Omron Sysmac Studio project Colorificio_End_Release (Sysmac Studio 1.30.0.17, StandardProject)
(* Comment update *)

# Controller PLC: NX1P2-9024DT1 version 1.40
Task PrimaryTask (priority 4, period or condition 2000): Program0
Library OmronLib_WC_Toolbox_V1_0 1.0.0 (contents left out)

TYPE S_Colori : STRUCT
    ALPHA : INT;
    RED : INT;
    GREEN : INT;
    BLU : INT;
    NOME : STRING[256];
END_STRUCT END_TYPE

VAR_GLOBAL
    SB0 : BOOL := False;  (* pulsante avvio ciclo automatico (NA); at BuiltInIO://cpu/#0/Input_Bit_00 *)
    SB1 : BOOL := True;  (* pulsante arresto ciclo automatico (NC); at BuiltInIO://cpu/#0/Input_Bit_01 *)
    SBE : BOOL := True;  (* pulsante arresto di emergenza (NC); at BuiltInIO://cpu/#0/Input_Bit_02 *)
    YVA : BOOL;  (* libera caricatore seconda latta (A-); at BuiltInIO://cpu/#0/Output_Bit_00 *)
    YVB : BOOL;  (* libera caricatore prima latta (B-); at BuiltInIO://cpu/#0/Output_Bit_01 *)
    YVC : BOOL;  (* scarico bilancia (C+); at BuiltInIO://cpu/#0/Output_Bit_02 *)
    KM1 : BOOL;  (* motore primo nastro; at BuiltInIO://cpu/#0/Output_Bit_09 *)
    KM2 : BOOL;  (* motore secondo nastro; at IOBus://unit#3/Output Bit 8 bits/Output Bit 00 *)
    YVD : BOOL;  (* scarico coperchiatrice (D+); at BuiltInIO://cpu/#0/Output_Bit_03 *)
    a0 : BOOL := False;  (* caricatore seconda latta libero (NA); at BuiltInIO://cpu/#0/Input_Bit_03 *)
    a1 : BOOL := True;  (* caricatore seconda latta bloccato (NA); at BuiltInIO://cpu/#0/Input_Bit_04 *)
    b0 : BOOL := False;  (* caricatore prima latta libero (NA); at BuiltInIO://cpu/#0/Input_Bit_05 *)
    b1 : BOOL := True;  (* caricatore prima latta bloccato (NA); at BuiltInIO://cpu/#0/Input_Bit_06 *)
    c0 : BOOL := True;  (* scaricatore bilancia rientrato (NA); at BuiltInIO://cpu/#0/Input_Bit_07 *)
    c1 : BOOL := False;  (* scaricatore bilancia esteso (NA); at BuiltInIO://cpu/#0/Input_Bit_08 *)
    d0 : BOOL := True;  (* scaricatore coperchiatrice rientrato (NA); at BuiltInIO://cpu/#0/Input_Bit_09 *)
    d1 : BOOL := False;  (* scaricatore coperchiatrice esteso (NA); at BuiltInIO://cpu/#0/Input_Bit_10 *)
    BIL : REAL;  (* bilancia/cella di carico (Grammi) *)
    YVBASE : BOOL;  (* eroga colorante base; at BuiltInIO://cpu/#0/Output_Bit_04 *)
    YVRED : BOOL;  (* eroga colorante rosso; at BuiltInIO://cpu/#0/Output_Bit_05 *)
    YVGREEN : BOOL;  (* eroga colorante verde; at BuiltInIO://cpu/#0/Output_Bit_06 *)
    YVBLU : BOOL;  (* eroga colorante blu; at BuiltInIO://cpu/#0/Output_Bit_07 *)
    YVSCARICO : BOOL;  (* eroga totale colore; at BuiltInIO://cpu/#0/Output_Bit_08 *)
    Tbase : TIME;  (* tempo carico base *)
    Trosso : TIME;  (* tempo carico rosso *)
    Tgreen : TIME;  (* tempo carico verde *)
    Tblu : TIME;  (* tempo carico blu *)
    BLW : BOOL := True;  (* livello riserva Base White (NA); at BuiltInIO://cpu/#0/Input_Bit_11 *)
    BLR : BOOL := True;  (* livello riserva Red (NA); at BuiltInIO://cpu/#0/Input_Bit_12 *)
    BLG : BOOL := True;  (* livello riserva Green (NA); at BuiltInIO://cpu/#0/Input_Bit_13 *)
    BLB : BOOL := True;  (* livello riserva Blu (NA); at IOBus://unit#1/Input Bit 8 bits/Input Bit 00 *)
    BC1 : BOOL := False;  (* presenza seconda latta sul caricatore (NA); at IOBus://unit#1/Input Bit 8 bits/Input Bit 03 *)
    BBIL : BOOL := False;  (* presenza sulla bilancia (NA); at IOBus://unit#1/Input Bit 8 bits/Input Bit 01 *)
    BCOP : BOOL := False;  (* presenza sulla coperchiatrice (NA); at IOBus://unit#1/Input Bit 8 bits/Input Bit 04 *)
    RichiestaValvolaBase : BOOL;  (* Devo aprire la valvola della Base? *)
    RichiestaValvolaRosso : BOOL;  (* Devo aprire la valvola del Rosso? *)
    RichiestaValvolaVerde : BOOL;  (* Devo aprire la valvola del Verde? *)
    RichiestaValvolaBlu : BOOL;  (* Devo aprire la valvola del Blu? *)
    RichiestaValvolaTramoggia : BOOL;  (* Devo aprire la valvola della Tramoggia? *)
    LevelToEjectBase : REAL := -1;  (* Quantità di base da far uscire *)
    LevelToEjectRosso : REAL := -1;  (* Quantità di rosso da far uscire *)
    LevelToEjectVerde : REAL := -1;  (* Quantità di verde da far uscire *)
    LevelToEjectBlu : REAL := -1;  (* Quantità di blu da far uscire *)
    ColorDone : BOOL := False;  (* Processo di riempimento del barattolo completo *)
    PHL_RiservaBase : BOOL;  (* Lampada mancanza di base; at IOBus://unit#3/Output Bit 8 bits/Output Bit 01 *)
    PHL_RiservaRosso : BOOL;  (* Lampada mancanza di rosso; at IOBus://unit#3/Output Bit 8 bits/Output Bit 02 *)
    PHL_RiservaVerde : BOOL;  (* Lampada mancanza di verde; at IOBus://unit#3/Output Bit 8 bits/Output Bit 03 *)
    PHL_RiservaBlu : BOOL;  (* Lampada mancanza di blu; at IOBus://unit#3/Output Bit 8 bits/Output Bit 04 *)
    PHL_YVScarico : BOOL;  (* Lampada valvola tramoggia aperta; at IOBus://unit#3/Output Bit 8 bits/Output Bit 05 *)
    PHL_KM : BOOL;  (* Lampada nastri in movimento; at IOBus://unit#3/Output Bit 8 bits/Output Bit 06 *)
    PHL_Emergenza : BOOL;  (* Lampada pulsante emergenza attivato; at IOBus://unit#3/Output Bit 8 bits/Output Bit 07 *)
    LivelloTramoggia : REAL := 0.0;
    PesoTramoggia : REAL := 0.0;
    BC0 : BOOL := False;  (* presenza prima latta sul caricatore (NA); at IOBus://unit#1/Input Bit 8 bits/Input Bit 02 *)
END_VAR

PROGRAM Program0
VAR
    TimerBase : TP;
    TimerRosso : TP;
    TimerVerde : TP;
    TimerBlu : TP;
    estimatedBase : TIME;
    estimatedRosso : TIME;
    estimatedVerde : TIME;
    estimatedBlu : TIME;
    Rosso : BOOL;
    Base : BOOL;
    Verde : BOOL;
    Blu : BOOL;
    Scarico : BOOL;
    estimatedScarico : TIME;
    Tscarico : TIME;  (* Tempo di uscita del contenuto della tramoggia *)
    TimerScarico : TP;
    AspettaSvuotamentoBlu : TP;
    AspettaSvuotamentoBlu1 : TON;
    estimatedSvuotamentoBlu : TIME;
    estimatedSvuotamentoBlu1 : TIME;
    AspettaSvuotamentoScarico : TP;
    estimatedSvuotamentoScarico : TIME;
    AspettaSvuotamentoScarico1 : TON;
    estimatedSvuotamentoScarico1 : TIME;
    DelayBase : TON;  (* Attivazione base in ritardo *)
    estimatedActValvolaBase : TIME;  (* Tempo rimanente all'attivazione della valvola della base *)
    Basse : BOOL;
END_VAR
VAR_EXTERNAL
    SB1 : BOOL;
    KM1 : BOOL;
    YVC : BOOL;
    BBIL : BOOL;
    c0 : BOOL;
    c1 : BOOL;
    KM2 : BOOL;
    SB0 : BOOL;
    SBE : BOOL;
    BIL : REAL;
    RichiestaValvolaBase : BOOL;
    RichiestaValvolaRosso : BOOL;
    RichiestaValvolaVerde : BOOL;
    RichiestaValvolaBlu : BOOL;
    YVBASE : BOOL;
    YVRED : BOOL;
    YVGREEN : BOOL;
    YVBLU : BOOL;
    Tbase : TIME;
    Trosso : TIME;
    Tgreen : TIME;
    Tblu : TIME;
    RichiestaValvolaTramoggia : BOOL;
    YVSCARICO : BOOL;
    ColorDone : BOOL;  (* Processo di riempimento del barattolo completo *)
    PHL_KM : BOOL;
    PHL_Emergenza : BOOL;
    PHL_YVScarico : BOOL;
    LevelToEjectBlu : REAL;
    LevelToEjectVerde : REAL;
    LevelToEjectRosso : REAL;
    LevelToEjectBase : REAL;
    LivelloTramoggia : REAL;
    PesoTramoggia : REAL;
    PHL_RiservaBase : BOOL;
    PHL_RiservaBlu : BOOL;
    PHL_RiservaVerde : BOOL;
    PHL_RiservaRosso : BOOL;
    BLB : BOOL;
    BLR : BOOL;
    BLW : BOOL;
    BLG : BOOL;
    BCOP : BOOL;
END_VAR
VAR
    _p1 : BOOL;
    _p2 : BOOL;
    _p3 : BOOL;
    _p4 : BOOL;
    _p5 : BOOL;
    _p6 : BOOL;
    _p7 : BOOL;
    _p8 : BOOL;
    _e9 : F_TRIG;
END_VAR

(* Section Section0: ladder, written here as Structured Text *)

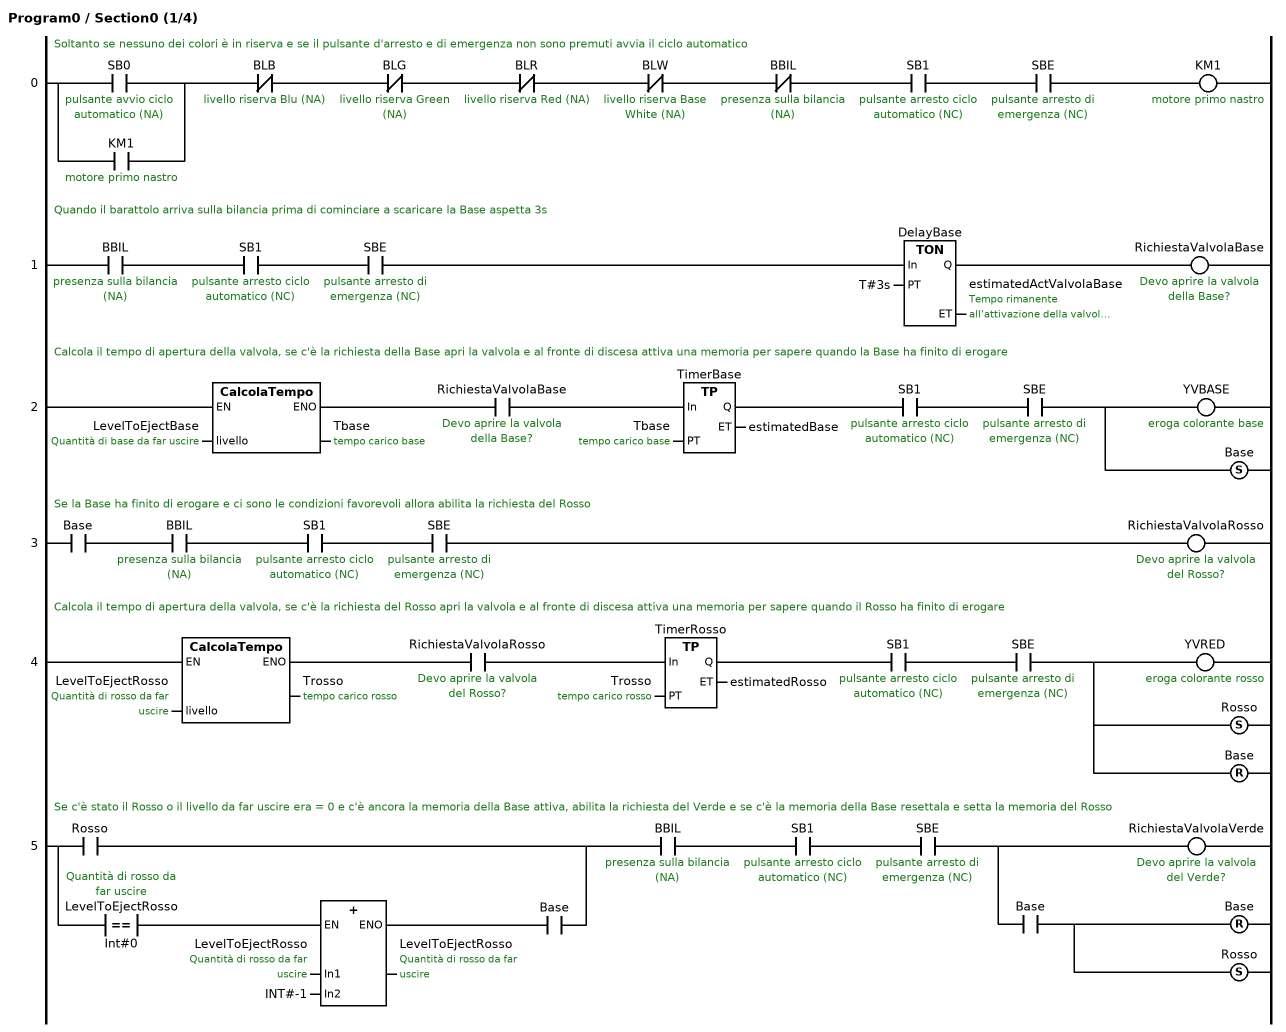
(* Rung 0: Soltanto se nessuno dei colori è in riserva e se il pulsante d'arresto e di emergenza non sono premuti avvia il ciclo automatico *)
KM1 := (SB0 OR KM1) AND NOT BLB AND NOT BLG AND NOT BLR AND NOT BLW AND NOT BBIL AND SB1 AND SBE;
(* Rung 1: Quando il barattolo arriva sulla bilancia prima di cominciare a scaricare la Base aspetta 3s *)
DelayBase(In := BBIL AND SB1 AND SBE, PT := T#3s, ET => estimatedActValvolaBase);
RichiestaValvolaBase := DelayBase.Q;
(* Rung 2: Calcola il tempo di apertura della valvola, se c'è la richiesta della Base apri la valvola e al fronte di discesa attiva una memoria per sapere quando la Base ha finito di erogare *)
Tbase := CalcolaTempo(livello := LevelToEjectBase);
TimerBase(In := RichiestaValvolaBase, PT := Tbase, ET => estimatedBase);
YVBASE := TimerBase.Q AND SB1 AND SBE;
IF TimerBase.Q AND SB1 AND SBE THEN Base := TRUE; END_IF;
(* Rung 3: Se la Base ha finito di erogare e ci sono le condizioni favorevoli allora abilita la richiesta del Rosso *)
RichiestaValvolaRosso := Base AND BBIL AND SB1 AND SBE;
(* Rung 4: Calcola il tempo di apertura della valvola, se c'è la richiesta del Rosso apri la valvola e al fronte di discesa attiva una memoria per sapere quando il Rosso ha finito di erogare *)
Trosso := CalcolaTempo(livello := LevelToEjectRosso);
TimerRosso(In := RichiestaValvolaRosso, PT := Trosso, ET => estimatedRosso);
YVRED := TimerRosso.Q AND SB1 AND SBE;
IF TimerRosso.Q AND SB1 AND SBE THEN
    Rosso := TRUE;
    Base := FALSE;
END_IF;
(* Rung 5: Se c'è stato il Rosso o il livello da far uscire era = 0 e c'è ancora la memoria della Base attiva, abilita la richiesta del Verde e se c'è la memoria della Base resettala e setta la memoria del Rosso *)
_p1 := LevelToEjectRosso = Int#0;
IF _p1 THEN LevelToEjectRosso := LevelToEjectRosso + (INT#-1); END_IF;
_p2 := (Rosso OR (_p1 AND Base)) AND BBIL AND SB1 AND SBE;
RichiestaValvolaVerde := _p2;
_p3 := _p2 AND Base;
IF _p3 THEN
    Base := FALSE;
    Rosso := TRUE;
END_IF;

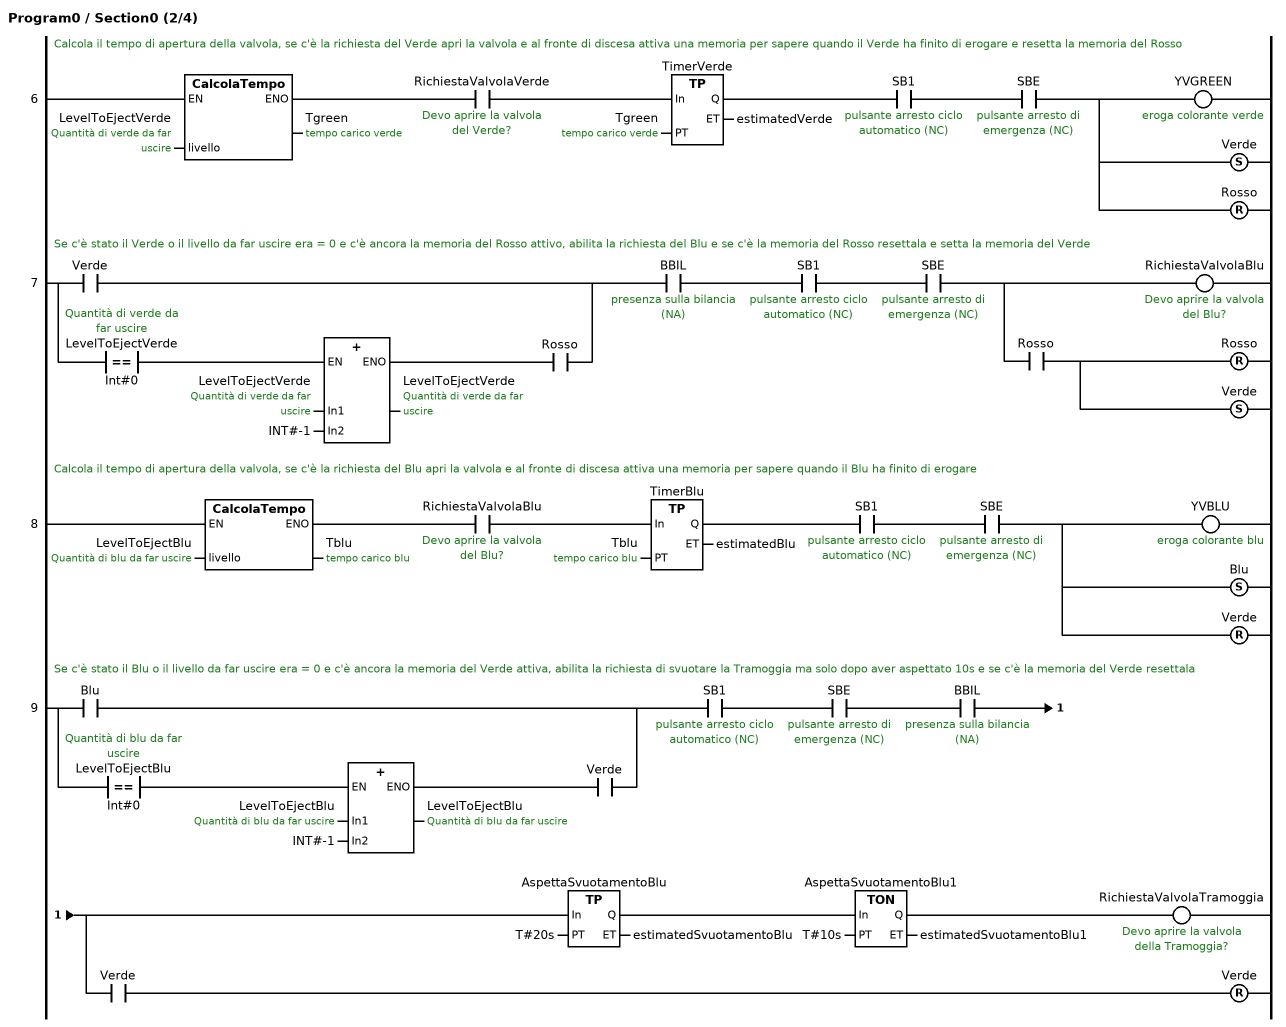
(* Rung 6: Calcola il tempo di apertura della valvola, se c'è la richiesta del Verde apri la valvola e al fronte di discesa attiva una memoria per sapere quando il Verde ha finito di erogare e resetta la memoria del Rosso *)
Tgreen := CalcolaTempo(livello := LevelToEjectVerde);
TimerVerde(In := RichiestaValvolaVerde, PT := Tgreen, ET => estimatedVerde);
YVGREEN := TimerVerde.Q AND SB1 AND SBE;
IF TimerVerde.Q AND SB1 AND SBE THEN
    Verde := TRUE;
    Rosso := FALSE;
END_IF;
(* Rung 7: Se c'è stato il Verde o il livello da far uscire era = 0 e c'è ancora la memoria del Rosso attivo, abilita la richiesta del Blu e se c'è la memoria del Rosso resettala e setta la memoria del Verde *)
_p4 := LevelToEjectVerde = Int#0;
IF _p4 THEN LevelToEjectVerde := LevelToEjectVerde + (INT#-1); END_IF;
_p5 := (Verde OR (_p4 AND Rosso)) AND BBIL AND SB1 AND SBE;
RichiestaValvolaBlu := _p5;
_p6 := _p5 AND Rosso;
IF _p6 THEN
    Rosso := FALSE;
    Verde := TRUE;
END_IF;
(* Rung 8: Calcola il tempo di apertura della valvola, se c'è la richiesta del Blu apri la valvola e al fronte di discesa attiva una memoria per sapere quando il Blu ha finito di erogare *)
Tblu := CalcolaTempo(livello := LevelToEjectBlu);
TimerBlu(In := RichiestaValvolaBlu, PT := Tblu, ET => estimatedBlu);
YVBLU := TimerBlu.Q AND SB1 AND SBE;
IF TimerBlu.Q AND SB1 AND SBE THEN
    Blu := TRUE;
    Verde := FALSE;
END_IF;
(* Rung 9: Se c'è stato il Blu o il livello da far uscire era = 0 e c'è ancora la memoria del Verde attiva, abilita la richiesta di svuotare la Tramoggia ma solo dopo aver aspettato 10s e se c'è la memoria del Verde resettala *)
_p7 := LevelToEjectBlu = Int#0;
IF _p7 THEN LevelToEjectBlu := LevelToEjectBlu + (INT#-1); END_IF;
_p8 := (Blu OR (_p7 AND Verde)) AND SB1 AND SBE AND BBIL;
AspettaSvuotamentoBlu(In := _p8, PT := T#20s, ET => estimatedSvuotamentoBlu);
AspettaSvuotamentoBlu1(In := AspettaSvuotamentoBlu.Q, PT := T#10s, ET => estimatedSvuotamentoBlu1);
RichiestaValvolaTramoggia := AspettaSvuotamentoBlu1.Q;
IF _p8 AND Verde THEN Verde := FALSE; END_IF;

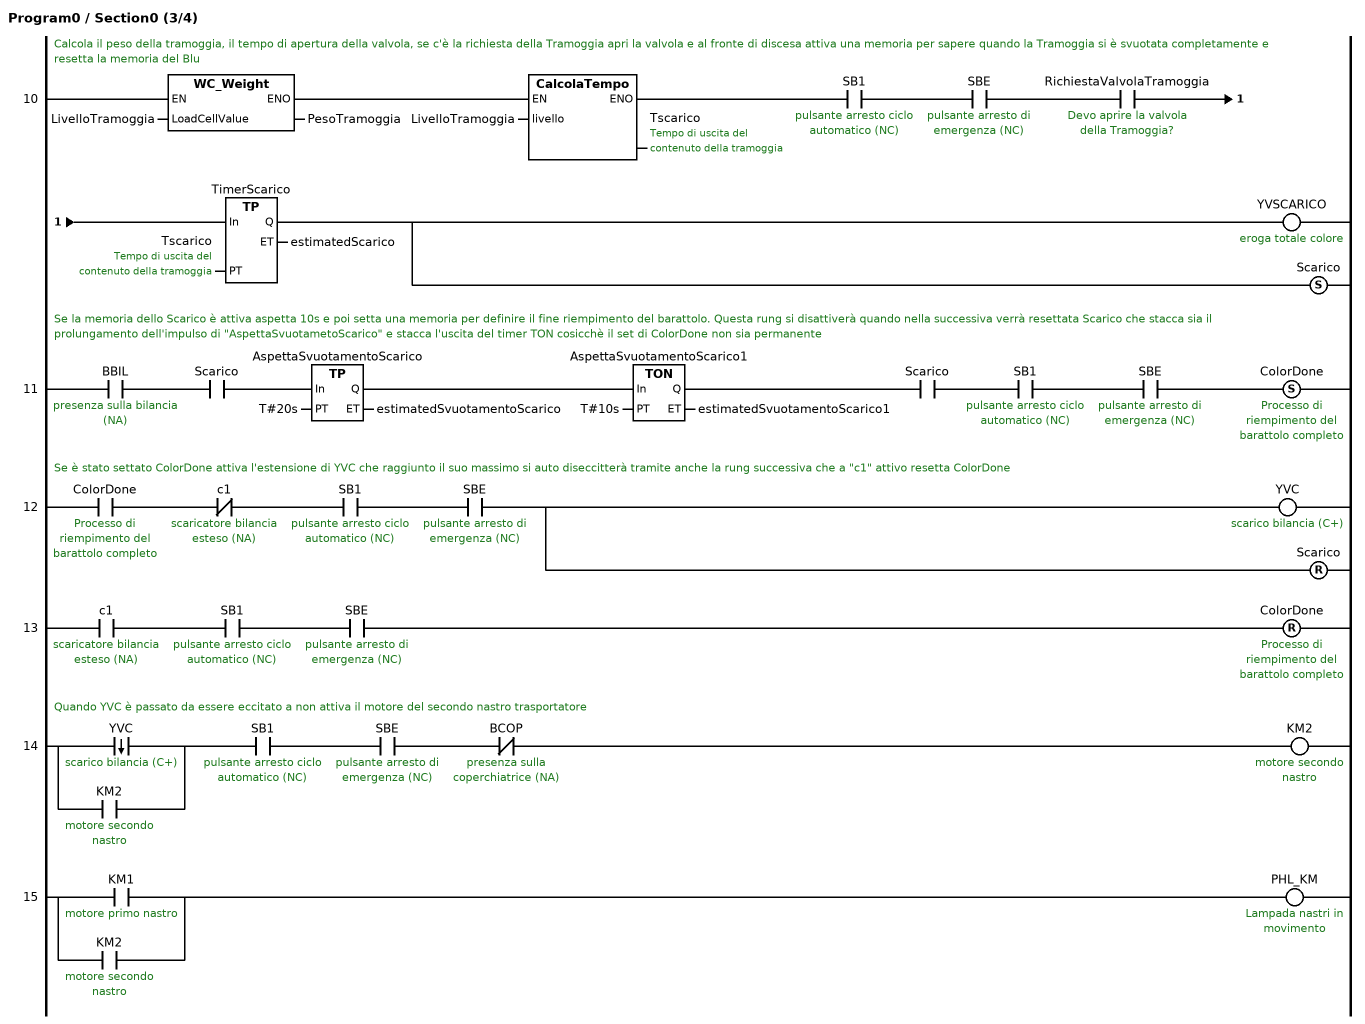
(* Rung 10: Calcola il peso della tramoggia, il tempo di apertura della valvola, se c'è la richiesta della Tramoggia apri la valvola e al fronte di discesa attiva una memoria per sapere quando la Tramoggia si è svuotata completamente e resetta la memoria del Blu *)
PesoTramoggia := WC_Weight(LoadCellValue := LivelloTramoggia);
Tscarico := CalcolaTempo(livello := LivelloTramoggia);
TimerScarico(In := SB1 AND SBE AND RichiestaValvolaTramoggia, PT := Tscarico, ET => estimatedScarico);
YVSCARICO := TimerScarico.Q;
IF TimerScarico.Q THEN Scarico := TRUE; END_IF;
(* Rung 11: Se la memoria dello Scarico è attiva aspetta 10s e poi setta una memoria per definire il fine riempimento del barattolo. Questa rung si disattiverà quando nella successiva verrà resettata Scarico che stacca sia il prolungamento dell'impulso di "AspettaSvuotametoScarico" e stacca l'uscita del timer TON cosicchè il set di ColorDone non sia permanente *)
AspettaSvuotamentoScarico(In := BBIL AND Scarico, PT := T#20s, ET => estimatedSvuotamentoScarico);
AspettaSvuotamentoScarico1(In := AspettaSvuotamentoScarico.Q, PT := T#10s, ET => estimatedSvuotamentoScarico1);
IF AspettaSvuotamentoScarico1.Q AND Scarico AND SB1 AND SBE THEN ColorDone := TRUE; END_IF;
(* Rung 12: Se è stato settato ColorDone attiva l'estensione di YVC che raggiunto il suo massimo si auto diseccitterà tramite anche la rung successiva che a "c1" attivo resetta ColorDone *)
YVC := ColorDone AND NOT c1 AND SB1 AND SBE;
IF ColorDone AND NOT c1 AND SB1 AND SBE THEN Scarico := FALSE; END_IF;
(* Rung 13 *)
IF c1 AND SB1 AND SBE THEN ColorDone := FALSE; END_IF;
(* Rung 14: Quando YVC è passato da essere eccitato a non attiva il motore del secondo nastro trasportatore *)
_e9(CLK := YVC);
KM2 := (_e9.Q OR KM2) AND SB1 AND SBE AND NOT BCOP;
(* Rung 15 *)
PHL_KM := KM1 OR KM2;

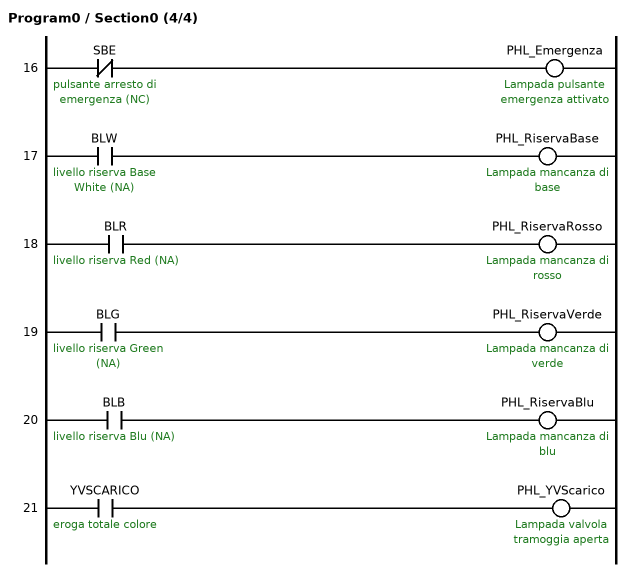
(* Rung 16 *)
PHL_Emergenza := NOT SBE;
(* Rung 17 *)
PHL_RiservaBase := BLW;
(* Rung 18 *)
PHL_RiservaRosso := BLR;
(* Rung 19 *)
PHL_RiservaVerde := BLG;
(* Rung 20 *)
PHL_RiservaBlu := BLB;
(* Rung 21 *)
PHL_YVScarico := YVSCARICO;
END_PROGRAM

FUNCTION CalcolaTempo : TIME
VAR
    Temporanea : REAL;
END_VAR
VAR_INPUT
    livello : REAL;
END_VAR
IF livello < 0 THEN
	CalcolaTempo := T#0s;
ELSE
	Temporanea := 0.2 ** 0.5; 
	Temporanea := Temporanea * 2 * livello;
	Temporanea := Temporanea ** 0.5;
	// Data la quantità di fluido da far uscire calcola il tempo che impiegherebbe supponendo che lo spazio da percorrere perchè il liquido superi la valvola sia di 20 cm = 0.2 m
	// Formula derivata dalla legge di Torricelli

	CalcolaTempo := NanoSecToTime(REAL_TO_INT(Temporanea) * 1000000000);
END_IF;
END_FUNCTION

FUNCTION WC_Weight : REAL
VAR_INPUT
    LoadCellValue : REAL;
END_VAR
// Il valore espresso è il peso in kili

IF LoadCellValue = 0 THEN
	WC_Weight := 0;
ELSE
	WC_Weight := LoadCellValue*0.03; // LoadCellValue = livello colore della tramoggia di pesatura
END_IF;
END_FUNCTION

# Device HMI (NA): not converted